(* IEC 61131-3 sources: codesys-build/examples/frame-assembly/src/framing/FB_FramingStation, 2 files *)

(* ---- declaration.st ---- *)
FUNCTION_BLOCK FB_FramingStation
VAR
	State : E_StationState := E_StationState.Idle;
	Completed : UDINT;
END_VAR

(* ---- FB_FramingStation.implementation.st ---- *)
CASE State OF
	E_StationState.Idle: State := E_StationState.Working;
	E_StationState.Working:
		Completed := Completed + 1;
		State := E_StationState.Idle;
END_CASE
